Fanuc KAREL source: ka00185.KL

-- PROVISIONAL review KL for V770-1; original PC SHA256 ac0ac9e70c1a8a3b16a5bf8022cf5964cfc1fe9da08fe0d63d5893efece30dc4
-- Incomplete behavior may be omitted. Consult companion uncertainty JSON. Do not deploy.
PROGRAM KA00185
%NOLOCKGROUP
-- UNRESOLVED_DECL SRC type=002018
-- UNRESOLVED_DECL DST type=002018
BEGIN
  -- UNRESOLVED_PC offsets 5-19; opcodes 22,22,1E
  -- UNRESOLVED_PC offsets 24-28; opcodes 7F
END KA00185
